TYPE TLoaderAxis :
	(
		LA_X := 0,
		LA_Y,
		LA_Z1,
		LA_Z2,
		LA_THETA
	);
END_TYPE

(* stored: Version 1.1.0.1, ProductVersion 3.1.4022.12
   DUT TLoaderAxis: Id {349e515f-508c-4028-b239-b641fa486901} *)
